FUNCTION_BLOCK LinearDA
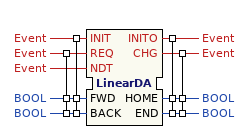
  EVENT_INPUT
    INIT WITH FWD, BACK;
    REQ WITH FWD, BACK;
    NDT;
  END_EVENT
  EVENT_OUTPUT
    INITO WITH HOME, END;
    CHG WITH HOME, END;
  END_EVENT
  VAR_INPUT
    FWD : BOOL;
    BACK : BOOL;
  END_VAR
  VAR_OUTPUT
    HOME : BOOL;
    END : BOOL;
  END_VAR
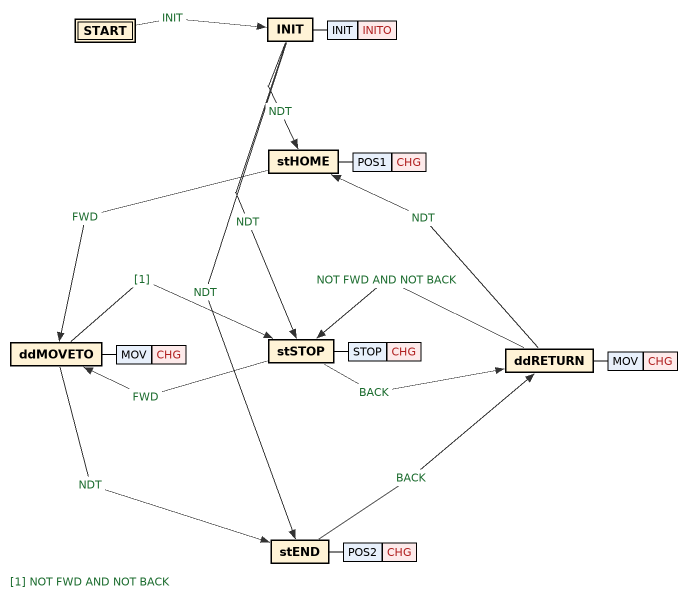
  EC_STATES
    START;
    INIT : INIT -> INITO;
    stHOME : POS1 -> CHG;
    stEND : POS2 -> CHG;
    ddMOVETO : MOV -> CHG;
    ddRETURN : MOV -> CHG;
    stSTOP : STOP -> CHG;
  END_STATES
  EC_TRANSITIONS
    START TO INIT := INIT;
    INIT TO stHOME := NDT;
    stHOME TO ddMOVETO := FWD;
    stEND TO ddRETURN := BACK;
    ddMOVETO TO stEND := NDT;
    ddRETURN TO stHOME := NDT;
    ddRETURN TO stSTOP := NOT FWD AND NOT BACK;
    stSTOP TO ddRETURN := BACK;
    stSTOP TO ddMOVETO := FWD;
    ddMOVETO TO stSTOP := NOT FWD AND NOT BACK;
    INIT TO stSTOP := NDT;
    INIT TO stEND := NDT;
  END_TRANSITIONS
  ALGORITHM INIT IN ST:
HOME := TRUE;
END := FALSE;
  END_ALGORITHM
  ALGORITHM POS1 IN ST:
HOME := TRUE;
END := FALSE;
  END_ALGORITHM
  ALGORITHM POS2 IN ST:
HOME := FALSE;
END := TRUE;
  END_ALGORITHM
  ALGORITHM MOV IN ST:
HOME := FALSE;
END := FALSE;
  END_ALGORITHM
  ALGORITHM STOP IN ST:
HOME := FALSE;
END := FALSE;
  END_ALGORITHM
END_FUNCTION_BLOCK
